// TIA Portal project "Asansör Projesi 2" (V17)

(* hardware
DEVICE "S71500/ET200MP-Station_1"  S7-1500 station
   slot 0: "Profilschiene_0"  6ES7 590-1***0-0AA0
   slot 1: "PLC_1"  CPU 1511-1 PN  6ES7 511-1AK00-0AB0  V1.8
   slot 2: "AI 8xU/I/RTD/TC ST_1"  AI 8xU/I/RTD/TC ST  6ES7 531-7KF00-0AB0  V2.0
   slot 3: "AI 8xU/I/RTD/TC ST_2"  AI 8xU/I/RTD/TC ST  6ES7 531-7KF00-0AB0  V2.0
   slot 4: "AI 8xU/I/RTD/TC ST_3"  AI 8xU/I/RTD/TC ST  6ES7 531-7KF00-0AB0  V2.0
   slot 5: "AI 8xU/I/RTD/TC ST_4"  AI 8xU/I/RTD/TC ST  6ES7 531-7KF00-0AB0  V2.0
   slot 6: "DI 16x24VDC BA_1"  DI 16x24VDC BA  6ES7 521-1BH10-0AA0  V1.0
*)

// ===== PLC "PLC_1"  CPU 1511-1 PN =====

VAR_GLOBAL   // PLC tag table "Standard-Variablentabelle"
   "Asansör 1.Kat" AT %E0.0 : Bool;
   "Asansör Yukarı" AT %A0.0 : Bool;
   "Asansör 2.Kat" AT %E0.1 : Bool;
   "1.Kat Yardımcı Kontak" AT %M0.0 : Bool;
   "Asansör 3.Kat" AT %I0.2 : Bool;
   "1.Kat Çağırma" AT %I0.3 : Bool;
   "2.Kat Çağırma" AT %I0.4 : Bool;
   "3.Kat Çağırma" AT %I0.5 : Bool;
   "2.Kat Yardımcı Kontak" AT %M0.1 : Bool;
   "3.Kat Yardımcı Kontak" AT %M0.2 : Bool;
   "1.Kat Sensör" AT %I0.7 : Bool;
   "Asansör Aşağı" AT %Q0.1 : Bool;
   "Asansör Yavaşlama" AT %Q0.2 : Bool;
   "2.Kat Sensör" AT %I1.0 : Bool;
   "3.Kat Sensör" AT %I1.1 : Bool;
   "3.Kat Frenleme Süresi" AT %T2 : Timer;
   "Acil Stop" AT %I0.6 : Bool;
   "Acil Stop Yardımcı Kontak 1" AT %M0.3 : Bool;
   "Acil Stop Yardımcı Kontak 2" AT %M0.4 : Bool;
   "1.Kat Frenleme Süresi" AT %T1 : Timer;
   "2.Kat Frenleme Süresi" AT %T0 : Timer;
   "Tag_3" AT %M0.5 : Bool;
   "Tag_4" AT %M0.6 : Bool;
END_VAR

// folder: System blocks/Program resources

DATA_BLOCK "T0"   // DB1
{ S7_Optimized_Access := 'TRUE' }
AUTHOR : Simatic
FAMILY : IEC
NAME : IEC_TMR
VERSION : 1.0
// stored: InstanceOfName IEC_TIMER
"IEC_TIMER"
BEGIN
END_DATA_BLOCK

DATA_BLOCK "T1"   // DB2
{ S7_Optimized_Access := 'TRUE' }
AUTHOR : Simatic
FAMILY : IEC
NAME : IEC_TMR
VERSION : 1.0
// stored: InstanceOfName IEC_TIMER
"IEC_TIMER"
BEGIN
END_DATA_BLOCK

DATA_BLOCK "T2"   // DB3
{ S7_Optimized_Access := 'TRUE' }
AUTHOR : Simatic
FAMILY : IEC
NAME : IEC_TMR
VERSION : 1.0
// stored: InstanceOfName IEC_TIMER
"IEC_TIMER"
BEGIN
END_DATA_BLOCK

// folder: (top level)

FUNCTION "MHJ-PLC-Lab-Function-S71500" : Void   // FC9000, SCL
{ S7_Optimized_Access := 'TRUE' }
VERSION : 0.1
   VAR_TEMP
      Value : Byte;
      ForCounter : Int;
   END_VAR
   VAR CONSTANT
      Value_01_DW : DWord := 16#1223_5486;
      Value_02_DW : DWord := 16#A6C9_D1F5;
   END_VAR
BEGIN

   #Value:=PEEK(area := 16#82,
        dbNumber := 0,
        byteOffset := 511);
   #Value := #Value + 1;

   POKE(area := 16#82,
        dbNumber := 0,
        byteOffset := 511,
        value := #Value);

   POKE(area := 16#82,
        dbNumber := 0,
        byteOffset := 1016,
        value := #Value_01_DW);
   POKE(area := 16#82,
        dbNumber := 0,
        byteOffset := 1020,
        value := #Value_02_DW);

   FOR #ForCounter := 0 TO 63 DO
       #Value:=PEEK(area := 16#1,
            dbNumber := 0,
            byteOffset := #ForCounter);
       POKE(area := 16#81,
            dbNumber := 0,
            byteOffset := #ForCounter,
            value := #Value);
   END_FOR;
   #Value := PEEK(area := 16#1,
                  dbNumber := 0,
                  byteOffset := 512);
   POKE(area := 16#82,
        dbNumber := 0,
        byteOffset := 512,
        value := #Value);
END_FUNCTION

ORGANIZATION_BLOCK "Main"   // OB1, LAD, ProgramCycle
TITLE = "Main Program Sweep (Cycle)"
{ S7_Optimized_Access := 'TRUE' }
VERSION : 0.1
   VAR_INPUT
      Initial_Call : Bool;   // Initial call of this OB
      Remanence : Bool;   // =True, if remanent data are available
   END_VAR
   VAR_TEMP   // added for the SCL form of the ladder/FBD networks
      _w1 : Bool;
      _w2 : Bool;
      _w3 : Bool;
      _w4 : Bool;
   END_VAR
BEGIN

REGION Network 1
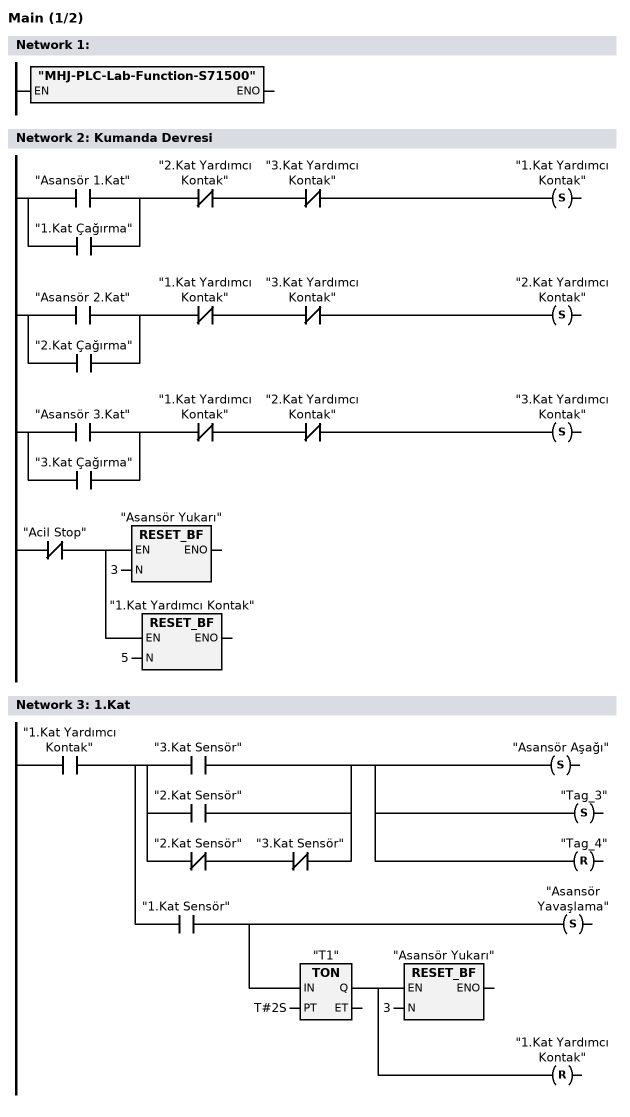
   RUNG wire#powerrail
      "MHJ-PLC-Lab-Function-S71500"()
   END_RUNG
   // the same network as SCL:
   "MHJ-PLC-Lab-Function-S71500"();
END_REGION

REGION Network 2: Kumanda Devresi
   // no SCL statement known for RBitfield: written as a call
   IF ("Asansör 1.Kat" OR "1.Kat Çağırma") AND NOT "2.Kat Yardımcı Kontak" AND NOT "3.Kat Yardımcı Kontak" THEN
       "1.Kat Yardımcı Kontak" := TRUE;
   END_IF;
   IF ("Asansör 2.Kat" OR "2.Kat Çağırma") AND NOT "1.Kat Yardımcı Kontak" AND NOT "3.Kat Yardımcı Kontak" THEN
       "2.Kat Yardımcı Kontak" := TRUE;
   END_IF;
   IF ("Asansör 3.Kat" OR "3.Kat Çağırma") AND NOT "1.Kat Yardımcı Kontak" AND NOT "2.Kat Yardımcı Kontak" THEN
       "3.Kat Yardımcı Kontak" := TRUE;
   END_IF;
   #_w1 := NOT "Acil Stop";
   IF #_w1 THEN
       RESET_BF(operand := "Asansör Yukarı", n := 3);
       RESET_BF(operand := "1.Kat Yardımcı Kontak", n := 5);
   END_IF;
END_REGION

REGION Network 3: 1.Kat
   // no SCL statement known for RBitfield: written as a call
   IF "1.Kat Yardımcı Kontak" AND ("3.Kat Sensör" OR "2.Kat Sensör" OR (NOT "2.Kat Sensör" AND NOT "3.Kat Sensör")) THEN
       "Asansör Aşağı" := TRUE;
       "Tag_3" := TRUE;
       "Tag_4" := FALSE;
   END_IF;
   #_w1 := "1.Kat Yardımcı Kontak" AND "1.Kat Sensör";
   IF #_w1 THEN "Asansör Yavaşlama" := TRUE; END_IF;
   "T1".TON(IN := #_w1, PT := T#2S);
   #_w2 := "T1".Q;
   IF #_w2 THEN
       RESET_BF(operand := "Asansör Yukarı", n := 3);
       "1.Kat Yardımcı Kontak" := FALSE;
   END_IF;
END_REGION

REGION Network 4: 2.Kat
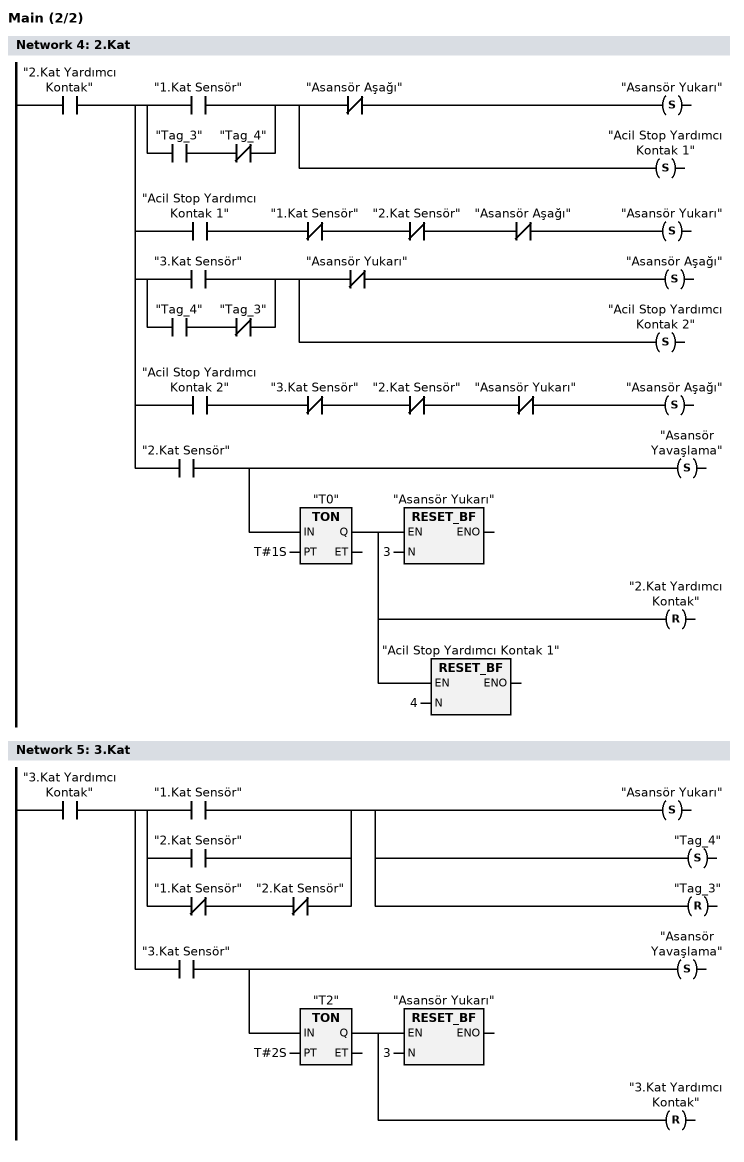
   // no SCL statement known for RBitfield: written as a call
   #_w1 := "2.Kat Yardımcı Kontak" AND ("1.Kat Sensör" OR ("Tag_3" AND NOT "Tag_4"));
   IF #_w1 AND NOT "Asansör Aşağı" THEN "Asansör Yukarı" := TRUE; END_IF;
   IF #_w1 THEN "Acil Stop Yardımcı Kontak 1" := TRUE; END_IF;
   IF "2.Kat Yardımcı Kontak" AND "Acil Stop Yardımcı Kontak 1" AND NOT "1.Kat Sensör" AND NOT "2.Kat Sensör" AND NOT "Asansör Aşağı" THEN
       "Asansör Yukarı" := TRUE;
   END_IF;
   #_w2 := "2.Kat Yardımcı Kontak" AND ("3.Kat Sensör" OR ("Tag_4" AND NOT "Tag_3"));
   IF #_w2 AND NOT "Asansör Yukarı" THEN "Asansör Aşağı" := TRUE; END_IF;
   IF #_w2 THEN "Acil Stop Yardımcı Kontak 2" := TRUE; END_IF;
   IF "2.Kat Yardımcı Kontak" AND "Acil Stop Yardımcı Kontak 2" AND NOT "3.Kat Sensör" AND NOT "2.Kat Sensör" AND NOT "Asansör Yukarı" THEN
       "Asansör Aşağı" := TRUE;
   END_IF;
   #_w3 := "2.Kat Yardımcı Kontak" AND "2.Kat Sensör";
   IF #_w3 THEN "Asansör Yavaşlama" := TRUE; END_IF;
   "T0".TON(IN := #_w3, PT := T#1S);
   #_w4 := "T0".Q;
   IF #_w4 THEN
       RESET_BF(operand := "Asansör Yukarı", n := 3);
       "2.Kat Yardımcı Kontak" := FALSE;
       RESET_BF(operand := "Acil Stop Yardımcı Kontak 1", n := 4);
   END_IF;
END_REGION

REGION Network 5: 3.Kat
   // no SCL statement known for RBitfield: written as a call
   IF "3.Kat Yardımcı Kontak" AND ("1.Kat Sensör" OR "2.Kat Sensör" OR (NOT "1.Kat Sensör" AND NOT "2.Kat Sensör")) THEN
       "Asansör Yukarı" := TRUE;
       "Tag_4" := TRUE;
       "Tag_3" := FALSE;
   END_IF;
   #_w1 := "3.Kat Yardımcı Kontak" AND "3.Kat Sensör";
   IF #_w1 THEN "Asansör Yavaşlama" := TRUE; END_IF;
   "T2".TON(IN := #_w1, PT := T#2S);
   #_w2 := "T2".Q;
   IF #_w2 THEN
       RESET_BF(operand := "Asansör Yukarı", n := 3);
       "3.Kat Yardımcı Kontak" := FALSE;
   END_IF;
END_REGION
END_ORGANIZATION_BLOCK